PROGRAM NCI
VAR
END_VAR

IF NOT PLC_CONSTANT.NCI_ACTIVE THEN RETURN; END_IF

END_PROGRAM

(* stored: Version 1.1.0.1, ProductVersion 3.1.4024.12
   POU NCI: Id {da86f3fe-4721-09d7-2e2d-987f1b92458d}, SpecialFunc None *)
